{attribute 'qualified_only'}
{attribute 'strict'}
TYPE State_Motor_Manipulator :
(
	OFF,
	INIT,
	RESET,
	READY,
	REF,
	PRODUCTION
);
END_TYPE

(* stored: Version 1.1.0.1, ProductVersion 3.1.4024.12
   DUT State_Motor_Manipulator: Id {3d27063f-58ae-4a6f-bdfd-9e989dca5f0a} *)
